Staubli VAL3: onF6Event.pgx

program onF6Event(bool& x_bSave[])
  local string l_sMessage
  local num i
  local num l_nSize
  local num l_nFound
  local string l_sEvent
  local bool l_bOk
  local string l_sButton[2]
  local num l_nItem
  local TrajectoryItem l_tTraj
begin
  // look if the bButton is enable
  if bButton[5]
    //
    // DELETE
    //
    call language:message(l_sMessage,80)
    call language:getYesNo(l_sButton)
    // ask the yes_no question
    call use:yes_no(l_sMessage,l_sButton,l_bOk)
    if l_bOk
      // look for select one
      call trajType:getSizeItem(false,l_nSize)
      l_nFound=0
      for i=0 to (l_nSize-1)
        if l_nSize>1
          call trajType:getTrajItem(l_tTraj,i)
          if find(l_tTraj.comment,"#")!=-1
            l_nFound=-1
            // delete both normal + user
            call trajType:deleteItem(i)
            i=i-1
            l_nSize=l_nSize-1
          endIf
        endIf
      endFor
      if l_nFound==0 and l_nSize>1
        l_nItem=nIndex
        call trajType:deleteItem(nIndex)
        nIndex=max(nIndex-1,0)
      endIf
      x_bSave=true
    endIf
  endIf
end
